FUNCTION_BLOCK FB_PIDControllerConsumer
VAR
    controller : B5PIDController_Plc.FB_PIDController;
    output : REAL;
END_VAR

controller(fError := 2.5);
output := controller.Step();

END_FUNCTION_BLOCK

(* stored: Version 1.1.0.1
   POU FB_PIDControllerConsumer: Id {7225539e-70b0-4b3f-b810-b7cb18fb252d}, SpecialFunc None *)
